(* Schneider Machine Expert - Basic project FlandersHVL-BaseSection-SingleController, file version 1.7.0.0 *)
(* ProjectInformations: Name=New project *)

HARDWARE
  Cpu 0: TM221M16R/G
  ModuleExtensionObject 0: TM2DDI32DK
  ModuleExtensionObject 1: TM2DDO32TK
  EthernetConfiguration: NetworkName=M221, IpAllocationMode=FixedAddress, IpAddress=0.0.0.0, SubnetMask=0.0.0.0
  SerialLineConfiguration: Baud=Baud19200, Parity=ParityEven, DataBits=DataBits8, StopBits=StopBits1, PhysicalMedium=PhysicalMediumRs485, TransmissionMode=TransmissionModeModbusRtu, SlaveId=1, Addressing=SlaveAddressing
  MastTask: UsePeriodScanMode=false, PeriodScan=100
  FastTask: Period=255
  CpuBehavior: StartingMode=StartAsPreviousState, AutoSaveRamOnEeprom=true, WatchdogPeriod=250

SYMBOLS  (address, symbol, comment, settings)
  %M0       STOP_ALARM
  %M1       RUN_STRIP_PULL
  %M2       EXTEND_CLAMP
  %M4       GLUE_TIMER_DN
  %TM0      STOP_ALARM_TIMER  [Preset=10, Base=OneSecond]
  %TM1      GLUE_TIMER  "Used to make sure glue doesn't go off the edge of the strip"  [Preset=3, Base=OneSecond]
  %I0.0     SYS_START
  %I0.1     SYS_RESET
  %I0.2     SYS_STOP
  %I0.3     SAFETY
  %I0.4     FILTER_AVAILABLE
  %I0.5     TAMPER_RET
  %I0.6     TAMPER_EXT
  %I0.7     VAC_CLAMP_RET
  %Q0.0     FAULT
  %Q0.1     GREEN_LIGHT
  %Q0.2     YELLOW_LIGHT
  %Q0.3     RED_LIGHT
  %Q0.4     ALARM
  %Q0.5     VAC_CLAMP
  %Q0.6     VACUUM
  %Q0.7     TAMPER
  %I1.0     VAC__CLAMP_EXT
  %I1.1     TAMP_MANUAL
  %I1.2     GLUE_EYE
  %I1.3     STRIP_AVAILABLE
  %Q2.0     STRIP_GUIDE
  %Q2.1     BOTTOM_STRIP_GLUE
  %Q2.2     TOP_STRIP_GLUE
  %Q2.3     PUSH_ROLLERS

POU Sstem Signals
  (* SectionNumber=1 *)

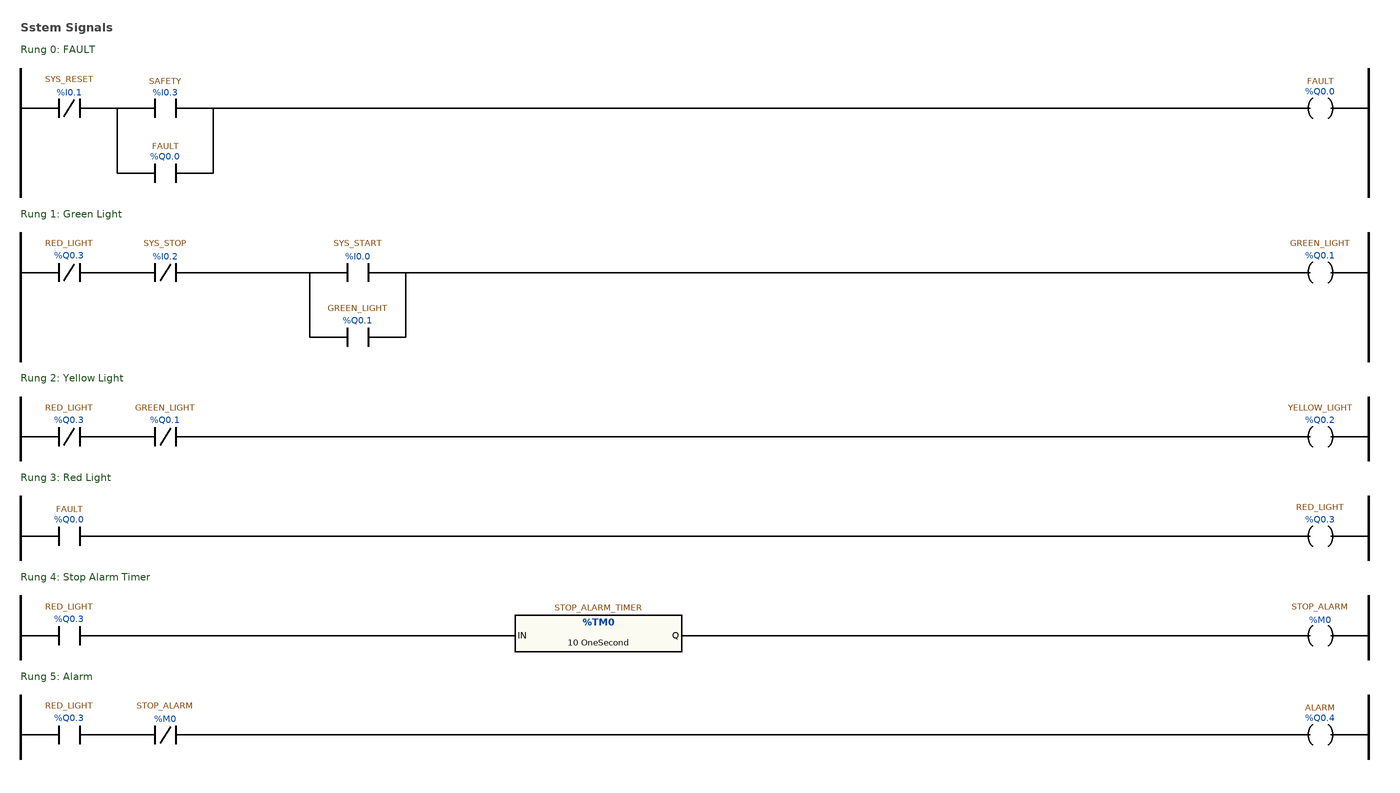

// Rung 0: FAULT
  LDN %I0.1               (* SYS_RESET *)
  AND( %I0.3              (* SAFETY *)
  OR %Q0.0                (* FAULT *)
  )
  ST %Q0.0                (* FAULT *)
  // as ST:
  //   FAULT := NOT SYS_RESET AND (SAFETY OR FAULT);

// Rung 1: Green Light
  LDN %Q0.3               (* RED_LIGHT *)
  ANDN %I0.2              (* SYS_STOP *)
  AND( %I0.0              (* SYS_START *)
  OR %Q0.1                (* GREEN_LIGHT *)
  )
  ST %Q0.1                (* GREEN_LIGHT *)
  // as ST:
  //   GREEN_LIGHT := NOT RED_LIGHT AND NOT SYS_STOP AND (SYS_START OR GREEN_LIGHT);

// Rung 2: Yellow Light
  LDN %Q0.3               (* RED_LIGHT *)
  ANDN %Q0.1              (* GREEN_LIGHT *)
  ST %Q0.2                (* YELLOW_LIGHT *)
  // as ST:
  //   YELLOW_LIGHT := NOT RED_LIGHT AND NOT GREEN_LIGHT;

// Rung 3: Red Light
  LD %Q0.0                (* FAULT *)
  ST %Q0.3                (* RED_LIGHT *)
  // as ST:
  //   RED_LIGHT := FAULT;

// Rung 4: Stop Alarm Timer
  BLK %TM0                (* STOP_ALARM_TIMER *)
  LD %Q0.3                (* RED_LIGHT *)
  IN
  OUT_BLK
  LD Q
  ST %M0                  (* STOP_ALARM *)
  END_BLK
  // as ST:
  //   STOP_ALARM_TIMER(IN := RED_LIGHT);
  //   STOP_ALARM := STOP_ALARM_TIMER.Q;

// Rung 5: Alarm
  LD %Q0.3                (* RED_LIGHT *)
  ANDN %M0                (* STOP_ALARM *)
  ST %Q0.4                (* ALARM *)
  // as ST:
  //   ALARM := RED_LIGHT AND NOT STOP_ALARM;

POU Strip Machine
  (* SectionNumber=2 *)

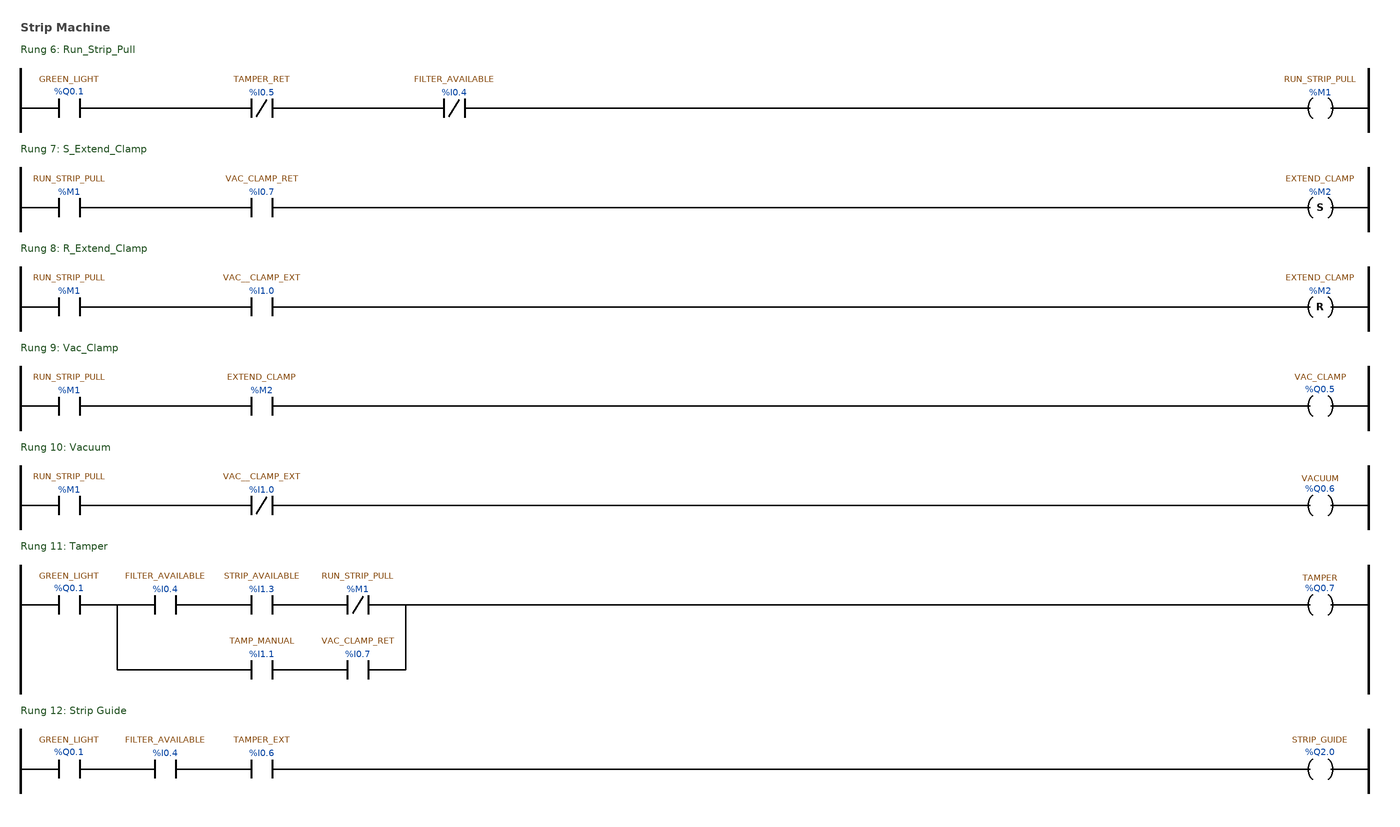

// Rung 6: Run_Strip_Pull
  LD %Q0.1                (* GREEN_LIGHT *)
  ANDN %I0.5              (* TAMPER_RET *)
  ANDN %I0.4              (* FILTER_AVAILABLE *)
  ST %M1                  (* RUN_STRIP_PULL *)
  // as ST:
  //   RUN_STRIP_PULL := GREEN_LIGHT AND NOT TAMPER_RET AND NOT FILTER_AVAILABLE;

// Rung 7: S_Extend_Clamp
  LD %M1                  (* RUN_STRIP_PULL *)
  AND %I0.7               (* VAC_CLAMP_RET *)
  S %M2                   (* EXTEND_CLAMP *)
  // as ST:
  //   IF RUN_STRIP_PULL AND VAC_CLAMP_RET THEN EXTEND_CLAMP := TRUE; END_IF;

// Rung 8: R_Extend_Clamp
  LD %M1                  (* RUN_STRIP_PULL *)
  AND %I1.0               (* VAC__CLAMP_EXT *)
  R %M2                   (* EXTEND_CLAMP *)
  // as ST:
  //   IF RUN_STRIP_PULL AND VAC__CLAMP_EXT THEN EXTEND_CLAMP := FALSE; END_IF;

// Rung 9: Vac_Clamp
  LD %M1                  (* RUN_STRIP_PULL *)
  AND %M2                 (* EXTEND_CLAMP *)
  ST %Q0.5                (* VAC_CLAMP *)
  // as ST:
  //   VAC_CLAMP := RUN_STRIP_PULL AND EXTEND_CLAMP;

// Rung 10: Vacuum
  LD %M1                  (* RUN_STRIP_PULL *)
  ANDN %I1.0              (* VAC__CLAMP_EXT *)
  ST %Q0.6                (* VACUUM *)
  // as ST:
  //   VACUUM := RUN_STRIP_PULL AND NOT VAC__CLAMP_EXT;

// Rung 11: Tamper
  LD %Q0.1                (* GREEN_LIGHT *)
  AND( %I0.4              (* FILTER_AVAILABLE *)
  AND %I1.3               (* STRIP_AVAILABLE *)
  ANDN %M1                (* RUN_STRIP_PULL *)
  OR( %I1.1               (* TAMP_MANUAL *)
  AND %I0.7               (* VAC_CLAMP_RET *)
  )
  )
  ST %Q0.7                (* TAMPER *)
  // as ST:
  //   TAMPER := GREEN_LIGHT AND (FILTER_AVAILABLE AND STRIP_AVAILABLE AND NOT RUN_STRIP_PULL OR TAMP_MANUAL AND VAC_CLAMP_RET);

// Rung 12: Strip Guide
  LD %Q0.1                (* GREEN_LIGHT *)
  AND %I0.4               (* FILTER_AVAILABLE *)
  AND %I0.6               (* TAMPER_EXT *)
  ST %Q2.0                (* STRIP_GUIDE *)
  // as ST:
  //   STRIP_GUIDE := GREEN_LIGHT AND FILTER_AVAILABLE AND TAMPER_EXT;

POU Glue Machine
  (* SectionNumber=3 *)

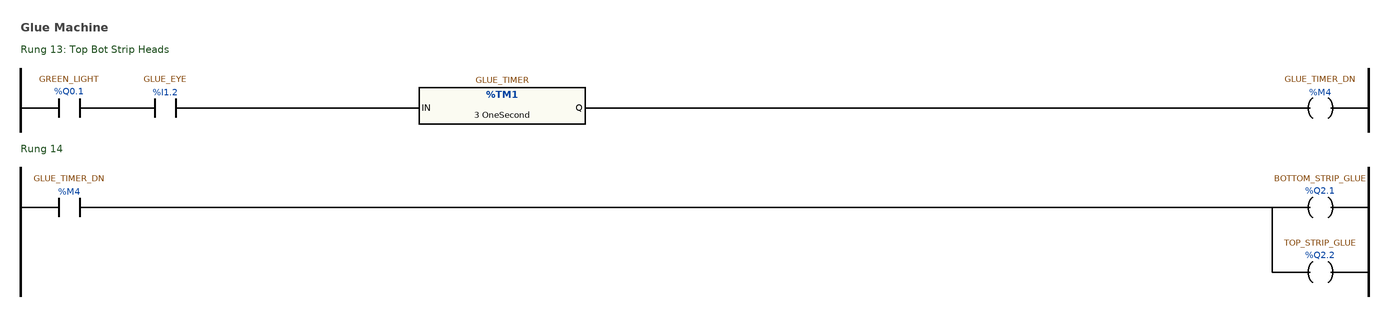

// Rung 13: Top Bot Strip Heads
  BLK %TM1                (* GLUE_TIMER *)
  LD %Q0.1                (* GREEN_LIGHT *)
  AND %I1.2               (* GLUE_EYE *)
  IN
  OUT_BLK
  LD Q
  ST %M4                  (* GLUE_TIMER_DN *)
  END_BLK
  // as ST:
  //   GLUE_TIMER(IN := GREEN_LIGHT AND GLUE_EYE);
  //   GLUE_TIMER_DN := GLUE_TIMER.Q;

// Rung 14
  LD %M4                  (* GLUE_TIMER_DN *)
  ST %Q2.1                (* BOTTOM_STRIP_GLUE *)
  ST %Q2.2                (* TOP_STRIP_GLUE *)
  // as ST:
  //   BOTTOM_STRIP_GLUE := GLUE_TIMER_DN;
  //   TOP_STRIP_GLUE := GLUE_TIMER_DN;
